PROGRAM MAIN
VAR
	// Variable for VLS upstream pressure bit
	{attribute 'pytmc' := '
	pv: EXT_PRESS_OK ;
	field: ZNAM NOT OK ;
	field: ONAM OK ;
	io: i ;
	'}
	bVLS_Press_OK : BOOL := FALSE; // TRUE : OK to open gate valve, FALSE : not OK to open gate valve
	
//	stPTM : ST_PfeifferControl;
//	fbPTM : FB_PTM_Pfeiffer;
END_VAR

(* Example main program to show how to incorporate the VLS vacuum program *)

PRG_VLS_VACUUM();

END_PROGRAM

(* stored: Version 1.1.0.1, ProductVersion 3.1.4022.18
   POU MAIN: Id {17e1a7f8-0f0e-4430-9e7a-0ad1f9ee68e0}, SpecialFunc None *)
